FUNCTION FahrenheitToCelsius : Celsius
VAR_INPUT
    temperature : Fahrenheit;
END_VAR

FahrenheitToCelsius.IOError := temperature.IOError;
FahrenheitToCelsius.WorkingCounterError := temperature.WorkingCounterError;
IF IsValid(temperature) THEN
    FahrenheitToCelsius._ := (temperature._ - 32) /  1.8;
END_IF

END_FUNCTION

(* stored: Version 1.1.0.1, ProductVersion 3.1.4024.4
   POU FahrenheitToCelsius: Id {675d4ac3-ebaa-4b9d-998c-2c3d2e5bd0ef}, SpecialFunc None *)
